FUNCTION TFMostUsedCode : INT
VAR_INPUT
	EnableCode : ARRAY [1..MAXFORMINGCODE*MAXFORMING] OF INT;
	UsedCode : POINTER TO ARRAY [1..MAXFORMINGCODE] OF INT;
END_VAR
VAR
	Code : INT;
	i : INT;
	j : INT;
	Counter : INT;
	MaxCounter : INT;
END_VAR

TFMostUsedCode := 0;
Code := 0;
MaxCounter := 0;

FOR i:=1 TO MAXFORMINGCODE*MAXFORMING DO
	IF EnableCode[i] > 0 THEN
		Counter := 0;
		FOR j:=1 TO MAXFORMINGCODE DO
			IF UsedCode^[j] = EnableCode[i] THEN
				Counter := Counter + 1;
			END_IF
		END_FOR
		IF Counter > MaxCounter THEN
			MaxCounter := Counter;
			Code := EnableCode[i];
		END_IF 
	END_IF
END_FOR

TFMostUsedCode := Code;

END_FUNCTION

(* stored: Version 1.1.0.1, ProductVersion 3.1.4024.11
   POU TFMostUsedCode: Id {5283495c-9a21-4494-bc64-61d9cc287282}, SpecialFunc None *)
